FUNCTION_BLOCK SysFunc1 (* Basic Function Block Type *)
  (* Standard: 61499-2 *)
  (* Version 0.0, 6/19/2016, Andrei, nxtControl GmbH, Template *)
  PACKAGE Main;
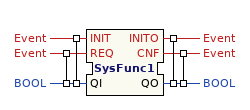
  EVENT_INPUT
    INIT WITH QI; (* Initialization Request *)
    REQ WITH QI; (* Normal Execution Request *)
  END_EVENT
  EVENT_OUTPUT
    INITO WITH QO; (* Initialization Confirm *)
    CNF WITH QO; (* Execution Confirmation *)
  END_EVENT
  VAR_INPUT
    QI : BOOL; (* Input event qualifier *)
  END_VAR
  VAR_OUTPUT
    QO : BOOL; (* Output event qualifier *)
  END_VAR
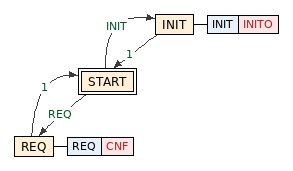
  EC_STATES
    START; (* Initial State *)
    INIT : INIT -> INITO; (* Initialization *)
    REQ : REQ -> CNF; (* Normal execution *)
  END_STATES
  EC_TRANSITIONS
    START TO INIT := INIT;
    INIT TO START := 1;
    START TO REQ := REQ;
    REQ TO START := 1;
  END_TRANSITIONS
  ALGORITHM INIT IN ST: (* Initialization algorithm *)
/*IF (onfloor0 OR onfloor1 OR onfloor2) = FALSE THEN
	RETURN;
END_IF;

IF onfloor0 THEN
	y:=0;
ELSIF onfloor1 THEN
	y:=1;
ELSIF onfloor2 THEN
	y:=2;
ELSE
	y:=-2;
END_IF;

IF gvl.doorclosed0 AND gvl.doorclosed1 AND gvl.doorclosed2 THEN
	allclosed := TRUE;
ELSE
	allclosed := FALSE;
END_IF;

IF y<>x THEN
	notx := TRUE;
ELSE
	notX:=FALSE;
END_IF;

// Liikkeelle lähtö
IF notX AND gvl.go AND allclosed THEN
	IF y>x THEN
		down:=TRUE;
	ELSE
		up:=TRUE;
	END_IF;
	closingX:=FALSE;
END_IF;

// Saavutaan matkan varrella kerrokseen 1 ja avataan ovi
IF (x<>1) AND gvl.onfloor1 AND (gvl.button1 OR gvl.call1 OR (timer1running)) THEN
	down:=FALSE;
	up:=FALSE;
	gvl.open1:=TRUE;
	t1.IN:=TRUE;
	t1.PT:=T#3S;
	t1();
	IF t1.Q THEN
		timer1running:=FALSE;
	ELSE
		timer1running:=TRUE;
	END_IF;
END_IF;

// Kerroksen 1 ovi kokonaan auki
IF t1.Q THEN
	t1.IN:=FALSE;
	t1();
	open1:=FALSE;
END_IF;

// Ollaan tai saavutaan kerrokseen x ja avataan ovi
IF (notX=FALSE) AND (closingX=FALSE) AND go THEN
	down:=FALSE;
	up:=FALSE;
	IF x=0 THEN
		gvl.open0:=TRUE;
	ELSIF x=1 THEN
		gvl.open1:=TRUE;
	ELSIF x=2 THEN
		gvl.open2:=TRUE;
	END_IF;
	tx.IN:=TRUE;
	tx.PT:=T#3S;
	tx();
	debug:=tx.ET;
	IF tx.Q THEN
		timer_Xrunning:=FALSE;
	ELSE
		timer_Xrunning:=TRUE;
	END_IF;

END_IF;

// Kerroksen x ovi kokonaan auki
IF tx.Q AND go THEN
	IF allclosed THEN
		go:=FALSE;
		tx.IN:=FALSE;
		tx();
	END_IF;
	closingX:=TRUE;
	IF x=0 THEN
		gvl.open0:=FALSE;
	ELSIF x=1 THEN
		gvl.open1:=FALSE;
	ELSIF x=2 THEN
		gvl.open2:=FALSE;
	END_IF;
END_IF;

IF go=FALSE THEN
	closingX:=FALSE;
END_IF*/;
  END_ALGORITHM
  ALGORITHM REQ IN ST: (* Normally executed algorithm *)
;
  END_ALGORITHM
END_FUNCTION_BLOCK
